{attribute 'qualified_only'}
{attribute 'strict'}
TYPE EFeedbackMsgAstrofan612 :
(		
	StateMsg := 1,
	StatusMsg := 2,
	IsAliveMsg := 3,
	CurrentSpeedMsg := 10,
	TemperatureMsg,
	WarningRaisedMsg := 20,
	AlarmRaisedMsg,
	CustomMsg := 50
);
END_TYPE

(* stored: Version 1.1.0.1, ProductVersion 3.1.4024.12
   DUT EFeedbackMsgAstrofan612: Id {91353fe0-fc1a-428c-82b3-bbc28d0512c1} *)
